VAR_GLOBAL CONSTANT
	MAX_AXES 		: INT := 5;
	MAX_AXIS_GROUPS	: INT := 1;
END_VAR

(* stored: Version 1.1.0.1, ProductVersion 3.1.0.36
   GVL Motion_Parameters: Id {8f7824a3-7360-418f-b75e-813d66c522a2}, ParameterList True *)
